(* IEC 61131-3 sources: Daniele1996.github.io/AUTOMATION_AND_SOFTWARE_DESIGN_PATTERN/AUTOMATION_STUDIO/Task1/Logical/Knife, 3 files *)

(* ---- Types.typ ---- *)
TYPE
	Cutter_States:
		(
		Cutter_ready_to_be_initialized,
		Cutter_initializing,
		Cutter_ready_to_be_enabled,
		Cutter_enabling,
		Cutter_ready_to_be_disabled,
		Cutter_disabling
	);
END_TYPE

(* ---- Main.st ---- *)
PROGRAM _INIT
	(* Insert code here *)

END_PROGRAM

PROGRAM _CYCLIC
	(* Insert code here *)

	CASE state OF

		Cutter_ready_to_be_initialized:
			IF Cutter_Handler.Initialize THEN
				Axis_Enable := TRUE;

				state := Cutter_initializing;
			END_IF;

		Cutter_initializing:
			IF NOT Axis_Enable THEN
				Cutter_Handler.Initialize := FALSE;

				state := Cutter_ready_to_be_enabled;
			END_IF;

		Cutter_ready_to_be_enabled:
			IF Cutter_Handler.Enable THEN
				CUTTER_DISTANCE := BELT_POSITION;
				Axis_Command := AXIS_MOVE_ADDITIVE;

				state := Cutter_enabling;
			END_IF;

		Cutter_enabling:
			IF Axis_Command_Executed THEN
				Cutter_Handler.Enable := FALSE;

				state := Cutter_ready_to_be_disabled;
			END_IF;

		Cutter_ready_to_be_disabled:
			IF Cutter_Handler.Disable THEN
				CUTTER_DISTANCE := - BELT_POSITION;
				Axis_Command := AXIS_MOVE_ADDITIVE;

				state := Cutter_disabling;
			END_IF;

		Cutter_disabling:
			IF Axis_Command_Executed THEN
				Cutter_Handler.Disable := FALSE;

				state := Cutter_ready_to_be_enabled;
			END_IF;

	END_CASE;

	Knife.Slave	:= ADR(gKnife);

	Knife.AxisEnable_in := Axis_Enable;
	Knife.AxisCommand := Axis_Command;

	Knife.Distance	:= CUTTER_DISTANCE;
	Knife.Velocity := CUTTER_VELOCITY;
	Knife.Acceleration	:= CUTTER_ACCELLERATION;
	Knife.Deceleration	:= CUTTER_DEACCELLERATION;

	Knife();

	Axis_Enable := Knife.AxisEnable_out;
	Axis_Command_Executed := Knife.CommandExecuted;
	CUTTER_POSITION	:= Knife.ActualPosition;
	CUTTER_ACTUAL_VELOCITY:= Knife.ActualVelocity;

	ComTCP_SimOutputs.Shaft_1_ACT_POS := CUTTER_POSITION;

END_PROGRAM

PROGRAM _EXIT
	(* Insert code here *)

END_PROGRAM

(* ---- Variables.var ---- *)
VAR
	Knife : gAxis;
END_VAR

VAR
	state: Cutter_States := Cutter_ready_to_be_initialized;
END_VAR

VAR
	Axis_Command : WORD := AXIS_NULL_COMMAND;
	Axis_Command_Executed : BOOL;
	Axis_Enable : BOOL;
END_VAR

VAR
	CUTTER_POSITION : REAL;
	CUTTER_ACTUAL_VELOCITY : REAL;
	CUTTER_ACCELLERATION : REAL := 400;
	CUTTER_DEACCELLERATION : REAL := 400;
	CUTTER_DISTANCE : REAL;
	BELT_POSITION: REAL := 100;
END_VAR

VAR CONSTANT
	AXIS_NULL_COMMAND : WORD := 0;
	AXIS_MOVE_VELOCITY : WORD := 1;
	AXIS_MOVE_ADDITIVE : WORD := 2;
	AXIS_STOP : WORD := 3;
END_VAR
